TYPE Point3D :
STRUCT
	X : LREAL;
	Y : LREAL;
	Z : LREAL;
END_STRUCT
END_TYPE

(* stored: Version 1.1.0.1
   DUT Point3D: Id {dde23c33-936e-0ad7-358b-807b7d4e9d3b} *)
